(* PLC project gas_plant.project, CODESYS CODESYS V3.5 SP14 *)
(* stored: creationDateTime 2024-10-22T09:14:15.6442521, modificationDateTime 2024-10-22T09:13:57.2609233 *)

{attribute 'qualified_only'}
{attribute 'strict'}
TYPE Facility : (kernel := 0, user := 1, mail := 2, system := 3, sec_1 := 4, syslogd := 5, printer := 6, network := 7, uucp := 8, clock_1 := 9, sec_2 := 10, ftp := 11, ntp := 12, audit := 13, alert := 14, clock_2 := 15, local0 := 16, local1 := 17, local2 := 18, local3 := 19, local4 := 20, local5 := 21, local6 := 22, local7 := 23);
END_TYPE

{attribute 'qualified_only'}
{attribute 'strict'}
TYPE Severity : (Emergency := 0, Alert := 1, Critical := 2, Error := 3, Warning := 4, Notice := 5, Info := 6, Debug := 7);
END_TYPE

FUNCTION SpacePadDay : STRING(3)
  VAR_INPUT
    input_int : UINT;
  END_VAR
  VAR
    temp_len : USINT;
  END_VAR

            SpacePadDay := UINT_TO_STRING(input_int);
temp_len := INT_TO_USINT(len(SpacePadDay));

IF temp_len = 1 THEN
	SpacePadDay := INSERT(SpacePadDay, ' ', 0);
END_IF

SpacePadDay := CONCAT(SpacePadDay, ' ');
          
END_FUNCTION

FUNCTION_BLOCK syslogMessage
  VAR_INPUT
    facility : UINT;
    severity : UINT;
    host : STRING(64);
    tag : STRING(48);
    msg : STRING(256);
  END_VAR
  VAR
    prival : USINT;
    t : ARRAY[0..31] OF BYTE;
    index : UINT;
    temp_str : STRING(8);
    send_result : POINTER TO RTS_IEC_RESULT;
    sock_result : POINTER TO RTS_IEC_RESULT;
    socket : RTS_IEC_HANDLE := 0;
    message : ARRAY[0..512] OF BYTE;
  END_VAR

            // SYSLOG-MSG      = HEADER SP STRUCTURED-DATA [SP MSG]
// HEADER          = PRI VERSION SP TIMESTAMP SP HOSTNAME SP APP-NAME SP PROCID SP MSGID

// PRI             = "<" PRIVAL ">"
// PRIVAL          = 1*3DIGIT ; range 0 .. 191
prival := INT_TO_USINT(SHL(facility, 3) + (severity AND 16#07));
index := 0;
temp_str := '<';
my_memcopy(ADR(message[index]), 1, ADR(temp_str));
index := index + 1;
temp_str := USINT_TO_STRING(prival);
my_memcopy(ADR(message[index]), len(temp_str), ADR(temp_str));
index := index + len(temp_str);
temp_str := '>';
my_memcopy(ADR(message[index]), 1, ADR(temp_str));
index := index + 1;


t := Timestamp();
my_memcopy(ADR(message[index]), 15, ADR(t));
index := index + 15;

temp_str := ' ';
my_memcopy(ADR(message[index]), 1, ADR(temp_str));
index := index + 1;

my_memcopy(ADR(message[index]), len(host), ADR(host));
index := index + len(host);

temp_str := ' ';
my_memcopy(ADR(message[index]), 1, ADR(temp_str));
index := index + 1;

my_memcopy(ADR(message[index]), len(tag), ADR(tag));
index := index + len(tag);

temp_str := ': ';
my_memcopy(ADR(message[index]), 2, ADR(temp_str));
index := index + 2;

my_memcopy(ADR(message[index]), len(msg), ADR(msg));
index := index + len(msg);

IF socket = 0 THEN
	socket := SysSockCreate(iAddressFamily:= SOCKET_AF_INET, diType:=SOCKET_DGRAM , diProtocol:= 0, pResult:= sock_result);
END_IF
	
SysSockSendToUdp(
	hSocketUdp:= socket, 
	diPort:= 514, 
	szDestAddress:= '192.168.95.5', 
	pbyData:= ADR(message), 
	diDataSize:= index, 
	pResult:= send_result);
          
END_FUNCTION_BLOCK

FUNCTION Timestamp : ARRAY[0..31] OF BYTE
  VAR
    t_stamp : SYSTIMEDATE;
    utc : UDINT;
    result : RTS_IEC_RESULT;
    index : USINT;
    temp_str : STRING(8);
    temp_len : USINT;
    months : ARRAY[1..12] OF STRING := ['Jan', 'Feb', 'Mar', 'Apr', 'May', 'Jun', 'Jul', 'Aug', 'Sep', 'Oct', 'Nov', 'Dec'];
  END_VAR

            
index := 0;
utc := SysTimeRtcGet(result);
SysTimeRtcConvertUtcToDate(dwTimestampUtc:= utc, pDate:= t_stamp);

temp_str := months[t_stamp.wMonth];
my_memcopy(ADR(Timestamp[index]), 3, ADR(temp_str));
index := index + 3;

temp_str := ' ';
my_memcopy(ADR(Timestamp[index]), 1, ADR(temp_str));
index := index + 1;



// DATE-MDAY       = 2DIGIT  ; 01-28, 01-29, 01-30, 01-31 based on month/year
temp_str := SpacePadDay(t_stamp.wDay);
my_memcopy(ADR(Timestamp[index]), 3, ADR(temp_str));
index := index + 3;

temp_str := ZeroPadInt(t_stamp.wHour, 2);
my_memcopy(ADR(Timestamp[index]), 2, ADR(temp_str));
index := index + 2;

temp_str := ':';
my_memcopy(ADR(Timestamp[index]), 1, ADR(temp_str));
index := index + 1;

// TIME-MINUTE     = 2DIGIT  ; 00-59
temp_str := ZeroPadInt(UINT_TO_USINT(t_stamp.wMinute), 2);
my_memcopy(ADR(Timestamp[index]), 2, ADR(temp_str));
index := index + 2;

temp_str := ':';
my_memcopy(ADR(Timestamp[index]), 1, ADR(temp_str));
index := index + 1;

// TIME-SECOND     = 2DIGIT  ; 00-59
temp_str := ZeroPadInt(UINT_TO_USINT(t_stamp.wSecond), 2);
my_memcopy(ADR(Timestamp[index]), 2, ADR(temp_str));
index := index + 2;
index := index + 1;
          
END_FUNCTION

FUNCTION ZeroPadInt : STRING(4)
  VAR_INPUT
    input_int : UINT;
    length : USINT;
  END_VAR
  VAR
    temp_str : STRING(4);
    temp_len : USINT;
    zeroes : USINT;
  END_VAR

            ZeroPadInt := UINT_TO_STRING(input_int);
temp_len := INT_TO_USINT(len(ZeroPadInt));

zeroes := length - temp_len;
WHILE zeroes > 0 DO
	zeroes := zeroes - 1;
	ZeroPadInt := INSERT(ZeroPadInt, '0', 0);
END_WHILE


          
END_FUNCTION

FUNCTION my_memcopy : UINT
  VAR_INPUT
    dest_ptr : POINTER TO BYTE;
    size : UINT;
    data_item : POINTER TO BYTE;
  END_VAR
  VAR
    index_pointer : POINTER TO BYTE;
    data_pointer : POINTER TO BYTE;
    i : UINT;
    copied : UINT := 0;
  END_VAR

            // Copyright 2022 Fortiphyd Logic Inc
// All rights reserved
//

index_pointer := dest_ptr;
data_pointer := data_item;
FOR i := 0 TO size DO
	index_pointer^ := data_pointer^;
	index_pointer := index_pointer + 1;
	data_pointer := data_pointer + 1;
	copied := copied + 1;
END_FOR
my_memcopy := copied;
RETURN;

          
END_FUNCTION

PROGRAM SyslogExamples
  VAR
    syslogMessage_0 : syslogMessage;
    max_safe_rpm : UINT := 1100;
    TON_0 : TON;
    system_bytes_rx : UDINT;
    network_rx1 : UDINT := 0;
    network_rx2 : UDINT := 0;
    bandwidth : UDINT;
    syslogMessage_1 : syslogMessage;
    previous_process_state : UINT := 0;
    current_process_state : UINT := 0;
    syslogMessage_2 : syslogMessage;
    state_changed : BOOL;
  END_VAR

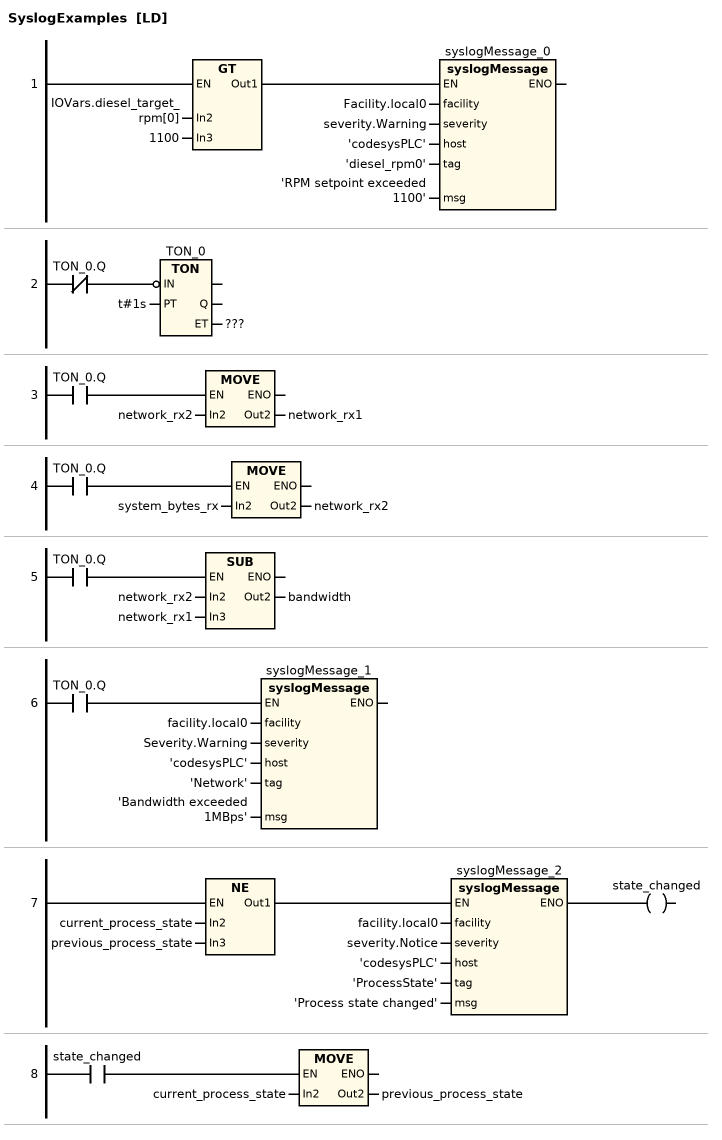
(* LD diagram, written out as Structured Text *)
(* Simple example of safety threshold alert *)

syslogMessage_0(EN := IOVars.diesel_target_rpm[0] > 1100, facility := Facility.local0, severity := severity.Warning, host := 'codesysPLC', tag := 'diesel_rpm0', msg := 'RPM setpoint exceeded 1100');
(* More complex example of watching network bytes received, 
you need to replace system_bytes_rx with your vendor's system call for bytes rx.

First, sample network bytes rx every 1 second and subtract previous
sample to get bytes/second. *)

TON_0(IN := NOT (NOT TON_0.Q), PT := t#1s, ET => ???);

IF TON_0.Q THEN network_rx1 := network_rx2; END_IF;

IF TON_0.Q THEN network_rx2 := system_bytes_rx; END_IF;

IF TON_0.Q THEN bandwidth := network_rx2 - network_rx1; END_IF;

syslogMessage_1(EN := TON_0.Q, facility := facility.local0, severity := Severity.Warning, host := 'codesysPLC', tag := 'Network', msg := 'Bandwidth exceeded 1MBps');
(* Simple example comparing the current process state with the previous one and logging the change.
The message string could include the state values using your system's string concat functions *)

syslogMessage_2(EN := current_process_state <> previous_process_state, facility := facility.local0, severity := severity.Notice, host := 'codesysPLC', tag := 'ProcessState', msg := 'Process state changed');
state_changed := syslogMessage_2.ENO;

IF state_changed THEN previous_process_state := current_process_state; END_IF;
END_PROGRAM
